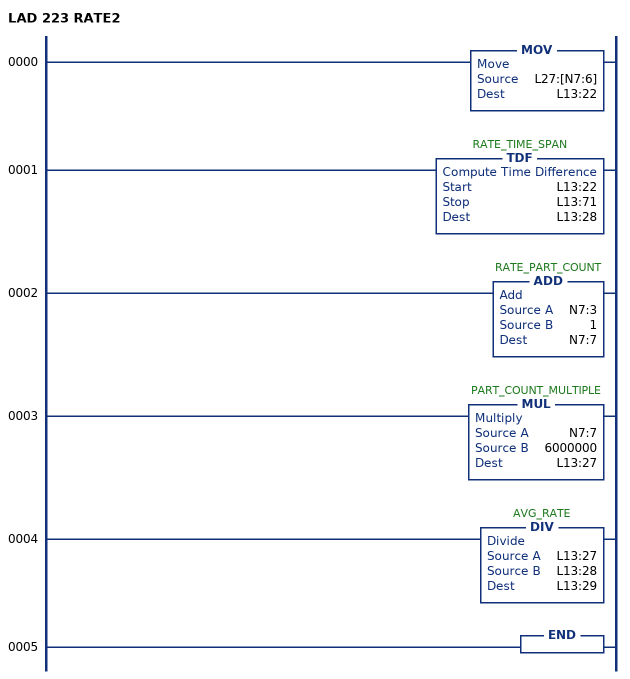
% Rung: 0 %
SOR MOV L27:[N7:6] L13:22 EOR
%   N7:6  OLDEST_TIME_INDEX %
% Rung: 1 %
SOR TDF L13:22 L13:71 L13:28 EOR
%   L13:71  HSC_TIME %
%   L13:28  RATE_TIME_SPAN %
% Rung: 2 %
SOR ADD N7:3 1 N7:7 EOR
%   N7:3  MAX_INDEX %
%   N7:7  RATE_PART_COUNT %
% Rung: 3 %
SOR MUL N7:7 6000000 L13:27 EOR
%   N7:7  RATE_PART_COUNT %
%   L13:27  PART_COUNT_MULTIPLE %
% Rung: 4 %
SOR DIV L13:27 L13:28 L13:29 EOR
%   L13:27  PART_COUNT_MULTIPLE %
%   L13:28  RATE_TIME_SPAN %
%   L13:29  AVG_RATE %
% Rung: 5 %
SOR END EOR

LADDER 224 "RESET RATE"
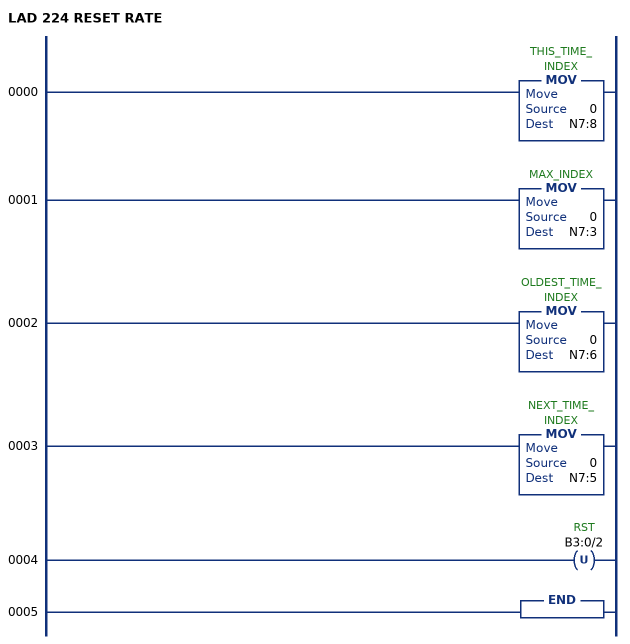
% Rung: 0 %
SOR MOV 0 N7:8 EOR
%   N7:8  THIS_TIME_INDEX %
% Rung: 1 %
SOR MOV 0 N7:3 EOR
%   N7:3  MAX_INDEX %
% Rung: 2 %
SOR MOV 0 N7:6 EOR
%   N7:6  OLDEST_TIME_INDEX %
% Rung: 3 %
SOR MOV 0 N7:5 EOR
%   N7:5  NEXT_TIME_INDEX %
% Rung: 4 %
SOR OTU B3:0/2 EOR
%   B3:0/2  RST %
% Rung: 5 %
SOR END EOR

OTHER DOCUMENTED ADDRESSES
  F8:12  "air pressure as float for hmi"
  I:0.0/0  BOTENCA
  I:0.0/1  BOTENCB
  I:0.0/3  INS1ACQ
  I:0.0/9  INS3ACQ
  I:0.0/10  INS3PASS
  I:0.0/11  INS3NG
  I:0.0/12  INS4ACQ
  I:0.0/13  INS4PASS
  I:0.0/14  INS4NG
  I:2.0/3  FRONT_ESTOP
  I:2.0/4  REAR_ESTOP
  I:2.0/5  FRONT_DOORS
  I:2.0/6  REAR_DOORS
  I:2.0/10  "spare"
  I:2.0/12  "spare"
  I:2.0/14  "spare"
  L42:0/1  "ps stop read (unused)"
  L42:1/2  "box full write (unused)"
  O:0.0/1  "spare? chute sensor?"
  O:0.0/4  TRIG_3  "spare"
  O:0.0/5  TRIG_4  "spare"
  O:0.0/9  "spare"
  O:0.0/10  "spare"
  O:0.0/11  "spare"
  O:3.0/0  "spare"
  O:3.0/2  "spare"
  O:3.0/3  LT_CTRN_RANGE_SELECT
  O:3.0/8  "spare"
  O:3.0/9  "spare"
  PFILE:6  "check for part jams"
  PFILE:10  "Bottom belt HSC"
  PFILE:12  "Top belt HSC"
  PFILE:123  "used for annylsys"
  Q2:55  END_OF_MAIN

COMMENTS NOT ATTACHED TO A CURRENT RUNG
  N17:8: ****************************************************************************************************************
    I can not find anywhere in the program where the "Test Spacing From Pickup to Trigger is activated indicating to me that this entire function must not be doing anything in this program at this time.
    ****************************************************************************************************************
  T20:2: The timer used to verify that the part that triggered the top laser optic has passed the bottom camer. needs to be count
  T20:2.ACC: This rung is starting a timer that should be activated directly before the laser optic part presense sensor on the top conveyer and should cause the top optic to be ignored if the bottom camera system didn't pass. however other arrangements must be made if the bottom camera isn't going to be used as is the case with a nut inspection.
  B22:0/0: ***********************
     Bottom Part Syncronizing Logic
    ***********************
    
    This is the point at the bottom of the top conveyor where the part jumps from the bottom conveyor.  This system will then track the part through the top system to the point of the laser optic in order to verify that the part in question has passed the bottom inspection.  I believe that we NEED to include FAILING inspections to eliminate the possibility of a out of position part from passing. LW 072010
  C5:4: tempory counting to verify pass part count with boxing part count.
  B23:0/0: Yet another bit shift load with data in the part position indicating that there was a bottom system part pass as well as a top system part present at this location.
    
    verified works w/bypassed 071910 and unbypassed 072010
  I:0.0/8: special rung for testing. This rung can simulate a pass signal. It will not be timed correctly.
  F8:13: *************************
    Loads Side Camera Passing data into a bit shift
    *************************
    
    loads passing data bit into passing data bit shift register at the part present cl.
  B3:7/9: ************************************
     The next 3 rungs appear to do nothing
    ***********************************
  B11:0/0: load part present bit shit with one shot data from the part present sensor
  RUNG000127-000009: multiply the current image acquire q by 11(ms) to get the current skip trigger delay
  RUNG000127-000010: time since oldest trigger
  RUNG000127-000012: trigger / capture part at trigger location
  RUNG000127-000015: time since last trigger
  RUNG000127-000017: remove used trigger bit
  B3:6/1: ***********************
    Part Width and  Location
    ***********************
    
    Calculates the position of parts on the top belt by measureing the part width by calculating the number of belt movement pulses that occure when the optic is blocked and then devides that in half and add that to the optic location in the part presnet bit shift when the top optic is cleared.
  B3:6/0: make a bit come on indicating that a part that passed the bottom camera is within  range when crossing the top camera.
  B9:0/[N7:47]: Remove any part present signals outside of expected location
  B9:0/[N7:50]: Remove any part present signals outside of expected location
  F19:0: Counter inside of a high speed counter interrupt counts the number of Bit Shifts that need to be processed in order to move the logic with the parts on the conveyor.
  F8:14: **************
    Bottom Top Camera Trigger
    *************
    
    Trigger Bottom Top Camera
  L13:104: Tracking error handler
  N10:4: test if boxing is connected
  T4:28: Check for buffer reset
  B3:11/3: After initial delay allow blow two start functioning
  RUNG000150-000041: transfer tracked part positon from trigger/acquire to the acquire/result
    capture acquire time
    reset process time
  RUNG000150-000039: Grab trigger/acquire position
    Grab acquire time
  RUNG000150-000038: acquire code
  RUNG000150-000035: fail count
  RUNG000150-000032: pass count
  RUNG000150-000025: pass code / Set pass bit in Bit Shift
    captures result position and processing time
    Unlatch pass bit
  RUNG000150-000018: pass, fail and acquire inputs
  RUNG000150-000016: wiped count
  RUNG000150-000014: clear data for time
  RUNG000150-000013: clear data for aquire time expired
  RUNG000150-000012: wipe stored part data if acq time expires
  RUNG000150-000011: trigger count
  L13:101: record the minimum time between triggers
  L14:5: on when ok to run, rear off turns both off
  L14:2: off when ok to run
  L14:3: off when ok to run
  L14:8: on when ok for run
  N7:76: removed relieance on trigger signal
  N197:20/0: Passes deformed head blowoff command to TOP PLC where solenoid output is located.
  L13:163: maximum average q
  L13:162: maximum q
  RUNG000141-000007: computer the time difference from the "pulled" data to the current time.
  RUNG000141-000006: convert offset data to a standard data because the TDF function can't handle offsets
  N7:50: ***********************************************************************************************************************************************************
    From top
    ***********************************************************************************************************************************************************
    
    removed relieance on trigger signal
  T4:20: Optic watchdog timers for faults
  B3:10/1: prevents momentary signals from box present sensor from tripping the logic for box not present
    
    This is in responce to a problem created by the sensor occasionally turning on as if no box was in its path when there is a box present.
  B3:6/2: IF PROCESSING FAULT OCURES AT COUNTER SENSOR; CLEAR THE BELT OF PASSING DATA
  L14:36: ****************  nEEDS fIXING  **********************
  L14:23: ****************  nEEDS fIXING  **********************
  RUNG000010-000018: Remove any part present signals outside of expected location
  RUNG000010-000014: ****
                      Zeros out the non passing part count when one passes
    ****
  T4:27: Check for buffer reset
  RUNG000125-000011: trigger count
  RUNG000125-000012: wipe stored part data if acq time expires
  RUNG000125-000013: clear data for aquire time expired
  RUNG000125-000014: clear data for time
  RUNG000125-000016: wiped count
  RUNG000125-000018: pass, fail and acquire inputs
  RUNG000125-000025: pass code / Set pass bit in Bit Shift
    captures result position and processing time
    Unlatch pass bit
  RUNG000125-000026: Grab trigger/acquire position
    Grab acquire time
  RUNG000125-000027: transfer tracked part positon from trigger/acquire to the acquire/result
    capture acquire time
    reset process time
  RUNG000125-000029: Set pass bit in Bit Shift
    captures result position and processing time
    Unlatch pass bit

REVISION NOTES
  13: updated count reset
  14: added io moduals
  15: multiple steps toward new hmi integration
  21: test

DATA TABLE (non-zero values as saved)
DATA B3
% B3:0 % 0X8191 0X0814 0XE040 0X8200 0XE100 0X8326 0X4605 0X0400 0X4007 0X0000
% B3:10 % 0X2041 0X0846 0X2000 0X0000 0X0000 0X0000 0X0000 0X0000 0X0000 0X0000
DATA T4
% .PRE .ACC %
% T4:1 % 200 200
% T4:2 % 333 50
% T4:3 % 300 0
% T4:4 % 400 0
% T4:5 % 250 0
% T4:6 % 10 32766
% T4:7 % 666 0
% T4:8 % 2 0
% T4:9 % 50 27
% T4:10 % 200 0
% T4:11 % 3 0
% T4:12 % 15 0
% T4:13 % 6 0
% T4:14 % 333 50
% T4:15 % 250 0
% T4:16 % 666 0
% T4:17 % 100 50
% T4:18 % 120 0
% T4:19 % 300 0
% T4:20 % 200 0
% T4:21 % 200 0
% T4:22 % 200 0
% T4:23 % 50 0
% T4:24 % 50 0
% T4:25 % 50 0
% T4:26 % 250 0
% T4:27 % 250 0
% T4:28 % 250 0
% T4:29 % 5000 0
% T4:30 % 50 50
% T4:31 % 20 0
% T4:32 % 69 0
DATA C5
% .PRE .ACC %
% C5:0 % 32766 0
DATA R6
% .LEN .POS %
% R6:0 % 20 0
% R6:1 % 3 0
% R6:2 % 3 0
% R6:3 % 3 0
% R6:4 % 1400 0
% R6:5 % 1400 0
% R6:6 % 1100 0
% R6:7 % 10 0
% R6:8 % 3 0
% R6:9 % 3 0
% R6:10 % 700 0
% R6:11 % 700 0
% R6:12 % 10 0
% R6:13 % 10 0
% R6:14 % 10 0
% R6:15 % 10 0
% R6:16 % 1100 0
% R6:17 % 700 0
% R6:18 % 700 0
% R6:19 % 10 0
DATA N7
% N7:0 % 1 9 6 0 13103 0 0 1 0 500
% N7:10 % 0 11 1 10 2 250 20 46 32766 10
% N7:20 % 666 333 32767 96 333 0 500 600 1000 1600
% N7:30 % 800 100 400 300 0 18021 2200 2200 777 0
% N7:40 % 333 0 1000 0 0 0 0 0 0 0
% N7:50 % 1236 0 175 16 0 1638 18021 0 12 0
% N7:60 % 1 32767 4012 20 31 0 0 15 30 20
% N7:70 % 0 21 23 27738 32767 0 122 0 16 0
% N7:80 % 0 6 95 0 0 0 5 500 0 0
% N7:90 % 2011 4 4 12 1 0 0 0 0 1600
% N7:100 % 1003 90 110 100 175 25 0 0 0 0
DATA F8
% F8:0 % 1 0 0 0 0
% F8:95 % 0 0 0 492 4.92
DATA B9
% B9:130 % 0X0000 0X0000 0X0000 0X0000 0X2000 0X0000 0X0000 0X0000 0X0000 0X8000
% B9:140 % 0X2480 0X0000 0X0000 0X0000 0X0000 0X0000 0X0000 0X0000 0X0000 0X0000
% B9:160 % 0X0000 0X0000 0X0000 0X0000 0X0000 0X0000 0X2000 0X0002 0X0000 0X0000
% B9:170 % 0X0000 0X0000 0X0000 0X2000 0X0000 0X0000 0X0000 0X0000 0X0000 0X0000
% B9:180 % 0X0000 0X0000 0X0000 0X0000 0X0000 0X0002 0X0000 0X0000 0X0000 0X0000
% B9:190 % 0X0010 0X0000 0X0000 0X0000 0X0000 0X0000 0X0000 0X0000 0X0000 0X0000
% B9:200 % 0X2B64 0X2B64 0X0000 0X0010 0X0000 0X2000 0X0000 0X0000 0X0000 0X0000
% B9:220 % 0X0000 0X0000 0X0000 0X0200 0X0000 0X0000 0X0000 0X0000 0X0000 0X0020
% B9:230 % 0X0040 0X0000 0X0000 0X0000 0X0000 0X0000 0X0000 0X0000 0X0000 0X0000
DATA B11
% B11:180 % 0X0000 0X8000 0X0000 0X0000 0X0000 0X0000 0X0000 0X0000 0X0000 0X0000
% B11:240 % 0X0000 0X0000 0X0000 0X4000 0X0000 0X0000 0X0000 0X0000 0X0000 0X0000
DATA B12
% B12:0 % 0X103D 0X0000 0X0000 0X0000 0X0000 0X0000 0X0000 0X0000 0X0000 0X0000
DATA L13
% L13:0 % 1 2600 0 -3550 1000
% L13:5 % 0 2 0 1162124017 1162124017
% L13:10 % 492 2 0 0 777
% L13:15 % 222509883 -2147483648 2147483647 335 477550
% L13:20 % 1578473548 77290636 -1971657207 335 2981458
% L13:25 % 998788400 36 6000000 -821784298 0
% L13:30 % 1575963506 0 36 2478822 1
% L13:35 % 478 1 1575963506 343 0
% L13:40 % 0 0 100 20 0
% L13:45 % 5 700 23 0 0
% L13:50 % 0 0 0 495000 60
% L13:55 % 53 9987884 342522 2600 444
% L13:60 % 3300 255 50 -1510198398 537159839
% L13:65 % 62 31 -640861925 -1444368236 -268230826
% L13:70 % 1501539718 1501539702 16 34549010 0
% L13:75 % 7 0 495000 -1510198339 -1510198385
% L13:80 % 46 537159849 150 0 200
% L13:85 % 12 200 45 26483 1000
% L13:90 % 26616 0 0 1000 0
% L13:95 % 60 99000 99000 25989 99000
% L13:100 % -1478910248 1 26 43 2025
% L13:105 % 1 0 1576329696 81 1576329679
% L13:110 % 17 40 10 537159595 537159593
% L13:115 % 537159600 7 4 537159596 1
% L13:120 % 0 50 0 30 49
% L13:125 % 164 19 155494060 137 155494060
% L13:130 % 1 1 0 2 1
% L13:135 % 0 1000 111 12 0
% L13:140 % 0 11 12 0 20
% L13:145 % 2568 1273 1284 111 111
% L13:150 % -1538760531 -1538760111 88 0 100
% L13:155 % 420 332 24 0 262301
% L13:160 % 3 7 4 395082 53203921
% L13:165 % 3 189116 95 13 8150
% L13:170 % 55946610 53 72 54 20
% L13:175 % 0 0 42 23 2021
% L13:180 % 176247033 25 99000 52866 644409
% L13:185 % 64 916459 92 627156 63
% L13:190 % 4 5 444 145219080 0
DATA F14
% F14:0 % 0 0 0 76 0
DATA N15
% N15:0 % 0 0 0 0 0 105 0 1356 0 10
DATA L16
% L16:0 % 8 14 11 0 20
% L16:5 % 250 5000 5000 182 19
% L16:10 % 1256 18 2045 6599584 98
% L16:15 % 99 0 0 0 0
DATA B17
% B17:60 % 0XC000 0X0000 0X0000 0X0000 0X0000 0X0000 0X0000 0X0000 0X0000 0X0000
% B17:100 % 0X0000 0X0000 0X0000 0X0000 0X0000 0X0000 0X0000 0X0000 0X1000 0X0000
% B17:110 % 0X4000 0X0000 0X0000 0X0000 0X0000 0X0000 0X0000 0X0000 0X0000 0X0000
% B17:120 % 0X0000 0X0000 0X0000 0X0000 0X0000 0X0000 0X0000 0X2000
DATA B18
% B18:60 % 0XC000 0X0000 0X0000 0X0000 0X0000 0X0000 0X0000 0X0000 0X0000 0X0000
% B18:100 % 0X0000 0X0000 0X0000 0X0000 0X0000 0X0000 0X0000 0X0000 0X0000 0X8240
% B18:110 % 0X0000 0X0400 0X0000 0X0000 0X0000 0X0000 0X0040 0X0000 0X0000 0X0010
% B18:120 % 0X0000 0X0000 0X0000 0X0000 0X0000 0X0000 0X0000 0X2000
DATA L23
% L23:0 % 65535 -65536 -65536 -65536 -65536
% L23:5 % -65536 -65536 2 65535 -65536
% L23:10 % -65536 0 17 10 17
% L23:15 % 0 0 0 0 8
% L23:20 % 0 -65536 -65536 -65536 -65536
% L23:25 % -65536 20 19 20 0
% L23:30 % 0 0 -65536 -65536 -65536
% L23:35 % -65536 -65536 -65536 -65536 -65536
% L23:40 % 16270 18414 0 63266 -65536
% L23:45 % 5062 0 0 0 0
% L23:50 % 0 -65536 -65536 17 -65536
% L23:55 % 33 5079 -65536 0 0
% L23:60 % 0 -65536 -65536 -65536 0
DATA L24
% L24:0 % -65536 122 -65536 222 -65536
% L24:5 % 65535 -65536 -65536 -65536 -65536
% L24:10 % 50 27 0 1 23
% L24:15 % 1198 1030 95 18 30
% L24:20 % 30 -65536 1226 -65536 -65536
% L24:25 % 222 1236 -65536 -65536 222
% L24:30 % 1466 27 10000 -65536 55
% L24:35 % 180 -65536 180 65535 101
% L24:40 % 101 1000 -65536 -65536 10
% L24:45 % 222 192 -65536 0 -65536
% L24:50 % -999 30 10000 65535 900
DATA L27
% L27:0 % -1971657207 -1971657007 -1971656807 -1971656606 -1971656401
% L27:5 % -1971656201 -1971656000 -1971655799 -1971655596 -1971655396
% L27:10 % -1971655194 -1971654993 -1971654791 -1971654582 -1971654385
% L27:15 % -1971654183 -1971653985 -1971653783 -1971653579 -1971653377
% L27:20 % -1971663352 -1971663156 -1971662956 -1971662653 -1971662549
% L27:25 % -1971662351 -1971662149 -1971661846 -1971661744 -1971661543
% L27:30 % -1971661337 -1971661136 -1971660937 -1971660738 -1971660532
% L27:35 % -1971660433 -1971660235 -1971660030 -1971659727 -1971659529
% L27:40 % -1971659327 -1971659126 -1971658920 -1971658721 -1971658518
% L27:45 % -1971658317 -1971658117 -1971657813 -1971657611 -1971657411
DATA L28
% L28:0 % 75067259 75067595 75068941 75069278 76457265
% L28:5 % 76457602 76458947 76459283 77288951 77289288
% L28:10 % 77290636 77290971 75035317 75035654 75037000
% L28:15 % 75037336 75038681 75039016 75040361 75040698
% L28:20 % 75042043 75042379 75043723 75044059 75045404
% L28:25 % 75045740 75047085 75047421 75048765 75049102
% L28:30 % 75050446 75050782 75052127 75052464 75053808
% L28:35 % 75054144 75055489 75055825 75057171 75057507
% L28:40 % 75058852 75059189 75060534 75060870 75062214
% L28:45 % 75062550 75063895 75064232 75065578 75065915
DATA L29
% L29:0 % 1578473548 1578473548 1578473548 1578473548 1578473548
% L29:5 % 1578473548 1578473548 1578473548 1578473548 1578473548
% L29:10 % 1578473548 1578473548 1578473548 1578473548 1578473548
% L29:15 % 1578473548 1578473548 1578473548 1578473548 1578473548
% L29:20 % 1578473548 1578473548 1578473548 1578473548 1578473548
% L29:25 % 1578473548 1578473548 1578473548 1578473548 1578473548
% L29:30 % 1578473548 1578473548 1578473548 1578473548 1578473548
% L29:35 % 1578473548 1578473548 1578473548 1578473548 1578473548
% L29:40 % 1578473548 1578473548 1578473548 1578473548 1578473548
% L29:45 % 1578473548 1578473548 1578473548 1578473548 1578473548
DATA L42
% L42:0 % 256 8 0 0 0
% L42:5 % 45 45 45 0 0
% L42:20 % 0 0 32766 32766 0
% L42:50 % 0 30
DATA L183
% L183:0 % 1427522383 1427522384 1 1000000000 0
% L183:5 % 7 26 55 0 0
DATA B185
% B185:0 % 0X0200 0X0001 0X0000 0X0000 0X0000 0X0000 0X0000 0X0000 0X0000 0X0000
DATA N186
% N186:0 % 100 0 0 0 0 0 0 0 0 0
DATA L187
% L187:0 % 34 26 497 0 0
DATA F188
% F188:0 % 0 66 11 44 29
DATA B189
% B189:0 % 0X00F1 0X0000 0X0000 0X0000 0X0000 0X0000 0X0000 0X0000 0X0000 0X0000
DATA L190
% L190:0 % 1 5 0 0 0
% L190:30 % 0 2 0 0 0
DATA B191
% B191:0 % 0X0000 0X0001 0X0000 0X0000 0X0000 0X0000 0X0000 0X0000 0X0000 0X0000
DATA L192
% L192:0 % -640861925 266932201 5055 0 0
% L192:5 % 1000000 0 999 999 8
% L192:10 % 0 0 1 78 17
% L192:15 % -1444152439 332250347 860888 77 0
% L192:20 % 180 39200000 0 0 0
DATA F193
% F193:0 % 0.3903424 0.315 0.022 6 0
% F193:5 % 0 0.02 0 0 419.7934
% F193:10 % 0.011 0.195 0.165 0.337 760
% F193:15 % -0.3382568 0.25 -0.08456421 696.6768 22827.31
DATA B195
% B195:90 % 0X0000 0X0000 0X0000 0X0000 0X0000 0X0000 0X0000 0X0040 0X0000 0X0000
DATA B196
% B196:0 % 0X0E24 0X9FF0 0X0005 0X0000 0X0000 0X0000 0X0000 0X0000 0X0000 0X0000
% B196:30 % 0XE800 0X9BFF 0XEBFF 0XFFDF 0XFFFF 0X0000 0X0000 0X0000 0X0000 0X0000
DATA N197
% N197:0 % 1560 150 500 2500 2500 14417 5555 0 200 0
% N197:10 % 4000 969 4 0 0 0 0 0 0 0
% N197:30 % 15 48 0 0 0 0 0 0 0 0
DATA B198
% B198:0 % 0X0009 0X0000 0X0000 0X0000 0X0000 0X0000 0X0000 0X0000 0X0000 0X0000
DATA L199
% L199:0 % 1 5571998 134 11 3579521
% L199:5 % 0 0 0 5 1064359
% L199:10 % 0 224 10256 556 0
% L199:15 % 0 0 0 278717848 518
% L199:20 % 28295 16430853 5001 5001 0
% L199:25 % 0 0 28329 1 3781224
% L199:30 % 21630086 251 3809367 15030467 111
% L199:35 % 555 555 0 0 0
DATA N200
% N200:0 % 2046 124 1 2047 1172 1594 1004 2045 2045 2045
% N200:10 % 0 0 0 1277 178 2046 1000 2045 2045 1218
% N200:20 % 1555 0 0 0 0 0 0 0 0 0
% N200:30 % 0 0 32767 0 0 0 0 0 0 0
DATA L201
% L201:0 % 20 40 40 -3011735 44
% L201:5 % 96629277 0 0 -3010662 0
% L201:10 % 0 0 0 327 43
% L201:15 % 0 43 0 43 36830
DATA B202
% B202:0 % 0X2241 0X0000 0X0001 0X0000 0X0000 0X0000 0X0000 0X0000 0X0000 0X0000
DATA N203
% N203:0 % 115 115 116 333 334 333 444 0 445 444
% N203:10 % 555 556 555 0 0 0 0 0 0 0
DATA L204
% L204:0 % 333 0 333 1362 124
% L204:5 % 2000 2000 462 222 0
% L204:10 % 0 0 0 1327077052 1327077052
% L204:15 % 1327077052 1327077052 1 0 0
% L204:20 % 0 0 33 0 0
% L204:30 % 33 0 0 0 0
DATA F205
% F205:0 % 25 66 0 66 0
